{attribute 'qualified_only'}
TYPE eEcatState :
(
	MASK          := 15,
	INIT          := 1, 
	PREOP         := 2,  
	BOOTSTRAP     := 3,  
	SAFEOP        := 4,  
	OP            := 8,  
	ERROR         := 16,  
	INVALID_VPRS  := 32,  
	INITCMD_ERROR := 48,  
	DISABLED      := 128 
)BYTE;
END_TYPE

(* stored: Version 1.1.0.1, ProductVersion 3.1.4024.10
   DUT eEcatState: Id {9950cb08-fabc-0a04-2fcc-9f1bc4d74f6a} *)
